// TIA Portal V20 export
TYPE "type_emRelations_em11_SoftCam"
// stored: Access Published, Namespace Unit1
   STRUCT
      spare { ExternalAccessible := 'False'; ExternalVisible := 'False'; ExternalWritable := 'False'} : Struct
         "00_position" : "LER_typeSoftCamPosition";
         "01_position" : "LER_typeSoftCamPosition";
         "02_position" : "LER_typeSoftCamPosition";
         "03_position" : "LER_typeSoftCamPosition";
         "04_posistion" { S7_SetPoint := 'True'} : "LER_typeSoftCamPosition";
         "05_posistion" { S7_SetPoint := 'True'} : "LER_typeSoftCamPosition";
         "06_posistion" { S7_SetPoint := 'True'} : "LER_typeSoftCamPosition";
         "07_posistion" { S7_SetPoint := 'True'} : "LER_typeSoftCamPosition";
         "08_posistion" { S7_SetPoint := 'True'} : "LER_typeSoftCamPosition";
         "09_posistion" { S7_SetPoint := 'True'} : "LER_typeSoftCamPosition";
         "10_posistion" { S7_SetPoint := 'True'} : "LER_typeSoftCamPosition";
         "11_posistion" { S7_SetPoint := 'True'} : "LER_typeSoftCamPosition";
         "12_posistion" { S7_SetPoint := 'True'} : "LER_typeSoftCamPosition";
         "13_posistion" { S7_SetPoint := 'True'} : "LER_typeSoftCamPosition";
         "14_posistion" { S7_SetPoint := 'True'} : "LER_typeSoftCamPosition";
         "15_posistion" { S7_SetPoint := 'True'} : "LER_typeSoftCamPosition";
      END_STRUCT;
   END_STRUCT;
END_TYPE
